FUNCTION_BLOCK FB_Impulsy
VAR_INPUT
	bWlacz									: BOOL;
	tZapalone								: TIME;
	tZgaszone								: TIME;
END_VAR
VAR_OUTPUT
END_VAR
VAR
	bWyjscie								: BOOL;
	tonZapalone								: TON;
	tonZgaszone								: TON;
END_VAR

IF (bWlacz) THEN
	tonZapalone (IN := NOT tonZgaszone.Q, PT := tZapalone);
	tonZgaszone (IN := tonZapalone.Q, PT := tZgaszone);
	
	IF (tonZapalone.Q) THEN
		bWyjscie								:= FALSE;
	ELSE
		bWyjscie								:= TRUE;
	END_IF
ELSE
	bWyjscie								:= FALSE;
END_IF

PROPERTY Wyjscie : BOOL
GET
Wyjscie									:= bWyjscie;
END_GET
END_PROPERTY

END_FUNCTION_BLOCK

(* stored: Version 1.1.0.1, ProductVersion 3.1.4024.11
   POU FB_Impulsy: Id {e5a1aeb6-776d-4742-99f2-eb32e9eabb99}, SpecialFunc None
   Property Wyjscie: Id {5b900922-ede1-4467-83da-7098377b5c69}
   Get Get: Id {322fb667-98e6-4751-897f-e369cd54b6f0} *)
